// TIA Portal project "2022.11.26-双轴组合搬运" (V17)
// Vorlageprojekt für das Buch mit Zielsystem S7-1200

(* hardware
DEVICE "S7-1200-Station_1"  S7-1200 Station
   slot 0: "Baugruppenträger_0"  Rack  V1.0
   slot 1: "PLC_1"  CPU 1214C DC/DC/DC  6ES7 214-1AG40-0XB0  V4.5
*)

// ===== PLC "PLC_1"  CPU 1214C DC/DC/DC =====

VAR_GLOBAL   // PLC tag table "Standard-Variablentabelle"
   "启动" AT %I1.2 : Bool;
   "暂停" AT %I1.3 : Bool;
   "启动灯" AT %Q1.1 : Bool;
   "暂停2" AT %M10.1 : Bool;
   "暂停灯" AT %Q1.2 : Bool;
   "启动(1)" AT %M10.0 : Bool;
   "上升沿暂存位" AT %M100.0 : Bool;
   "生成器1" AT %Q1.3 : Bool;
   "生成器2" AT %Q1.4 : Bool;
   "传送带1" AT %Q0.3 : Bool;
   "传送带2" AT %Q0.6 : Bool;
   "感应器1" AT %I0.3 : Bool;
   "上升沿暂存位(1)" AT %M100.2 : Bool;
   "感应器2" AT %I0.6 : Bool;
   "缩回1" AT %Q0.4 : Bool;
   "缩回2" AT %Q0.7 : Bool;
   "上升沿暂存位（2）" AT %M100.3 : Bool;
   "Tag_1" AT %M100.1 : Bool;
   "下降沿暂存位（1）" AT %M100.4 : Bool;
   "下降沿暂存位（2）" AT %M100.5 : Bool;
   "缩回感应" AT %I0.4 : Bool;
   "缩回感应2" AT %I0.7 : Bool;
   "拿下降" AT %Q0.1 : Bool;
   "拿下降感应" AT %I0.1 : Bool;
   "拿吸" AT %Q0.2 : Bool;
   "拿吸感应" AT %I0.2 : Bool;
   "拿有物" AT %M10.2 : Bool;
   "拿伸出" AT %Q0.0 : Bool;
   "拿伸出感应" AT %I0.0 : Bool;
   "拿放中" AT %M10.3 : Bool;
   "完成放物" AT %M10.5 : Bool;
   "完成拿放" AT %M10.6 : Bool;
   "上升1" AT %Q0.5 : Bool;
   "上升2" AT %Q1.0 : Bool;
   "上升感应1" AT %I0.5 : Bool;
   "上升感应2" AT %I1.0 : Bool;
   "计数" AT %M10.7 : Bool;
   "下降沿暂存位" AT %M100.6 : Bool;
   "计数(1)" AT %QD30 : DWord;
   "数据清零" AT %I1.4 : Bool;
   "清零灯" AT %Q1.5 : Bool;
END_VAR

// folder: System blocks/Program resources

DATA_BLOCK "T0"   // DB1
{ S7_Optimized_Access := 'TRUE' }
AUTHOR : Simatic
FAMILY : IEC
NAME : IEC_TMR
VERSION : 1.0
// stored: InstanceOfName IEC_TIMER
"IEC_TIMER"
BEGIN
END_DATA_BLOCK

DATA_BLOCK "T1"   // DB2
{ S7_Optimized_Access := 'TRUE' }
AUTHOR : Simatic
FAMILY : IEC
NAME : IEC_TMR
VERSION : 1.0
// stored: InstanceOfName IEC_TIMER
"IEC_TIMER"
BEGIN
END_DATA_BLOCK

DATA_BLOCK "T2"   // DB3
{ S7_Optimized_Access := 'TRUE' }
AUTHOR : Simatic
FAMILY : IEC
NAME : IEC_TMR
VERSION : 1.0
// stored: InstanceOfName IEC_TIMER
"IEC_TIMER"
BEGIN
END_DATA_BLOCK

DATA_BLOCK "T3"   // DB4
{ S7_Optimized_Access := 'TRUE' }
AUTHOR : Simatic
FAMILY : IEC
NAME : IEC_TMR
VERSION : 1.0
// stored: InstanceOfName IEC_TIMER
"IEC_TIMER"
BEGIN
END_DATA_BLOCK

DATA_BLOCK "T4"   // DB5
{ S7_Optimized_Access := 'TRUE' }
AUTHOR : Simatic
FAMILY : IEC
NAME : IEC_TMR
VERSION : 1.0
// stored: InstanceOfName IEC_TIMER
"IEC_TIMER"
BEGIN
END_DATA_BLOCK

DATA_BLOCK "T5"   // DB6
{ S7_Optimized_Access := 'TRUE' }
AUTHOR : Simatic
FAMILY : IEC
NAME : IEC_TMR
VERSION : 1.0
// stored: InstanceOfName IEC_TIMER
"IEC_TIMER"
BEGIN
END_DATA_BLOCK

DATA_BLOCK "T6"   // DB7
{ S7_Optimized_Access := 'TRUE' }
AUTHOR : Simatic
FAMILY : IEC
NAME : IEC_TMR
VERSION : 1.0
// stored: InstanceOfName IEC_TIMER
"IEC_TIMER"
BEGIN
END_DATA_BLOCK

// folder: (top level)

FUNCTION "MHJ-PLC-Lab-Function-S71200" : Void   // FC9000, SCL
{ S7_Optimized_Access := 'TRUE' }
VERSION : 0.1
   VAR_TEMP
      rdTimeReturn : Int;
      outputTime : DTL;
      SyncVal : Byte;
      forVal : Int;
      forVal_2 : Int;
      Value : Byte;
   END_VAR
   VAR CONSTANT
      CompVal : Byte := 16#34;
      Value_01 : Byte := 16#11;
      Value_01_DW : DWord := 16#A165_D992;
      Value_02_DW : DWord := 16#58BE_4401;
   END_VAR
BEGIN

   #Value:=PEEK(area := 16#82,
        dbNumber := 0,
        byteOffset := 511);
   #Value := #Value + 1;

   POKE(area := 16#82,
        dbNumber := 0,
        byteOffset := 511,
        value := #Value);

   POKE(area:=16#81,
        dbNumber:=0,
        byteOffset:=1016,
        value:=#Value_01_DW);
   POKE(area := 16#81,
        dbNumber := 0,
        byteOffset := 1020,
        value := #Value_02_DW);

   POKE(area := 16#81,
        dbNumber := 0,
        byteOffset := 511,
        value := B#16#00);

   FOR #forVal := 0 TO 120 DO
       FOR #forVal_2:=0 TO 10 DO
           #rdTimeReturn:=RD_SYS_T(#outputTime);
           #rdTimeReturn := WR_SYS_T(#outputTime);
           #rdTimeReturn := RD_SYS_T(#outputTime);
           #rdTimeReturn := WR_SYS_T(#outputTime);
       END_FOR;
       #SyncVal:= PEEK(area := 16#81,
                      dbNumber := 0,
                      byteOffset := 511);
       IF #SyncVal = #CompVal THEN
          GOTO M_1;
       END_IF;
   END_FOR;
   RETURN;

   M_1:
   POKE(area := 16#81,
        dbNumber := 0,
        byteOffset := 511,
        value := B#16#0);
END_FUNCTION

ORGANIZATION_BLOCK "Main"   // OB1, LAD, ProgramCycle
TITLE = "Main Program Sweep (Cycle)"
{ S7_Optimized_Access := 'TRUE' }
VERSION : 0.1
   VAR_INPUT
      Initial_Call : Bool;   // Initial call of this OB
      Remanence : Bool;   // =True, if remanent data are available
   END_VAR
   VAR_TEMP   // added for the SCL form of the ladder/FBD networks
      _w1 : Bool;
      _w2 : Bool;
      _w3 : Bool;
      _w4 : Bool;
   END_VAR
BEGIN

REGION Network 1
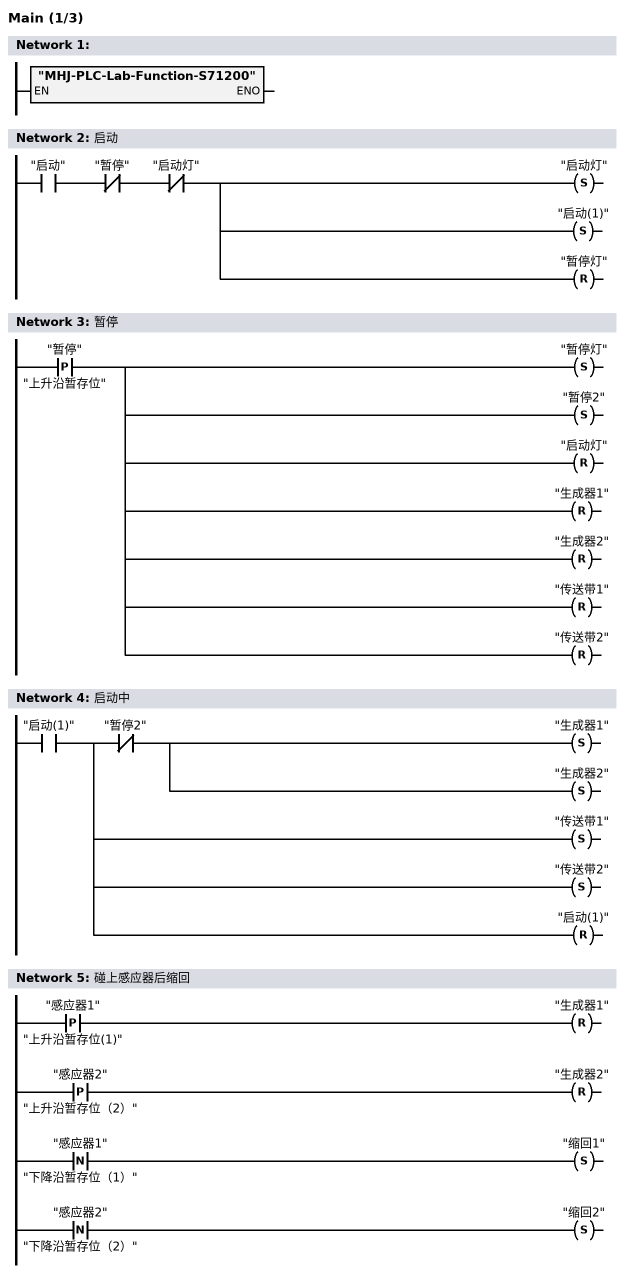
   RUNG wire#powerrail
      "MHJ-PLC-Lab-Function-S71200"()
   END_RUNG
   // the same network as SCL:
   "MHJ-PLC-Lab-Function-S71200"();
END_REGION

REGION Network 2: 启动
   RUNG wire#powerrail
      Contact( "启动" )
      I_Contact( "暂停" )
      I_Contact( "启动灯" )
      wire#w1
      S_Coil( "启动灯" )
   END_RUNG
   RUNG wire#w1
      S_Coil( "启动(1)" )
   END_RUNG
   RUNG wire#w1
      R_Coil( "暂停灯" )
   END_RUNG
   // the same network as SCL:
   #_w1 := "启动" AND NOT "暂停" AND NOT "启动灯";
   IF #_w1 THEN
       "启动灯" := TRUE;
       "启动(1)" := TRUE;
       "暂停灯" := FALSE;
   END_IF;
END_REGION

REGION Network 3: 暂停
   RUNG wire#powerrail
      P_Contact(operand := "暂停", bit := "上升沿暂存位")
      wire#w1
      S_Coil( "暂停灯" )
   END_RUNG
   RUNG wire#w1
      S_Coil( "暂停2" )
   END_RUNG
   RUNG wire#w1
      R_Coil( "启动灯" )
   END_RUNG
   RUNG wire#w1
      R_Coil( "生成器1" )
   END_RUNG
   RUNG wire#w1
      R_Coil( "生成器2" )
   END_RUNG
   RUNG wire#w1
      R_Coil( "传送带1" )
   END_RUNG
   RUNG wire#w1
      R_Coil( "传送带2" )
   END_RUNG
   // the same network as SCL:
   #_w1 := "暂停" AND NOT "上升沿暂存位";   // rising edge of "暂停"
   "上升沿暂存位" := "暂停";
   IF #_w1 THEN
       "暂停灯" := TRUE;
       "暂停2" := TRUE;
       "启动灯" := FALSE;
       "生成器1" := FALSE;
       "生成器2" := FALSE;
       "传送带1" := FALSE;
       "传送带2" := FALSE;
   END_IF;
END_REGION

REGION Network 4: 启动中
   RUNG wire#powerrail
      Contact( "启动(1)" )
      wire#w1
      I_Contact( "暂停2" )
      wire#w2
      S_Coil( "生成器1" )
   END_RUNG
   RUNG wire#w2
      S_Coil( "生成器2" )
   END_RUNG
   RUNG wire#w1
      S_Coil( "传送带1" )
   END_RUNG
   RUNG wire#w1
      S_Coil( "传送带2" )
   END_RUNG
   RUNG wire#w1
      R_Coil( "启动(1)" )
   END_RUNG
   // the same network as SCL:
   IF "启动(1)" AND NOT "暂停2" THEN
       "生成器1" := TRUE;
       "生成器2" := TRUE;
   END_IF;
   IF "启动(1)" THEN
       "传送带1" := TRUE;
       "传送带2" := TRUE;
       "启动(1)" := FALSE;
   END_IF;
END_REGION

REGION Network 5: 碰上感应器后缩回
   RUNG wire#powerrail
      P_Contact(operand := "感应器1", bit := "上升沿暂存位(1)")
      R_Coil( "生成器1" )
   END_RUNG
   RUNG wire#powerrail
      P_Contact(operand := "感应器2", bit := "上升沿暂存位（2）")
      R_Coil( "生成器2" )
   END_RUNG
   RUNG wire#powerrail
      N_Contact(operand := "感应器1", bit := "下降沿暂存位（1）")
      S_Coil( "缩回1" )
   END_RUNG
   RUNG wire#powerrail
      N_Contact(operand := "感应器2", bit := "下降沿暂存位（2）")
      S_Coil( "缩回2" )
   END_RUNG
   // the same network as SCL:
   #_w1 := "感应器1" AND NOT "上升沿暂存位(1)";   // rising edge of "感应器1"
   "上升沿暂存位(1)" := "感应器1";
   IF #_w1 THEN "生成器1" := FALSE; END_IF;
   #_w2 := "感应器2" AND NOT "上升沿暂存位（2）";   // rising edge of "感应器2"
   "上升沿暂存位（2）" := "感应器2";
   IF #_w2 THEN "生成器2" := FALSE; END_IF;
   #_w3 := NOT "感应器1" AND "下降沿暂存位（1）";   // falling edge of "感应器1"
   "下降沿暂存位（1）" := "感应器1";
   IF #_w3 THEN "缩回1" := TRUE; END_IF;
   #_w4 := NOT "感应器2" AND "下降沿暂存位（2）";   // falling edge of "感应器2"
   "下降沿暂存位（2）" := "感应器2";
   IF #_w4 THEN "缩回2" := TRUE; END_IF;
END_REGION

REGION Network 6: 缩回后拿下将
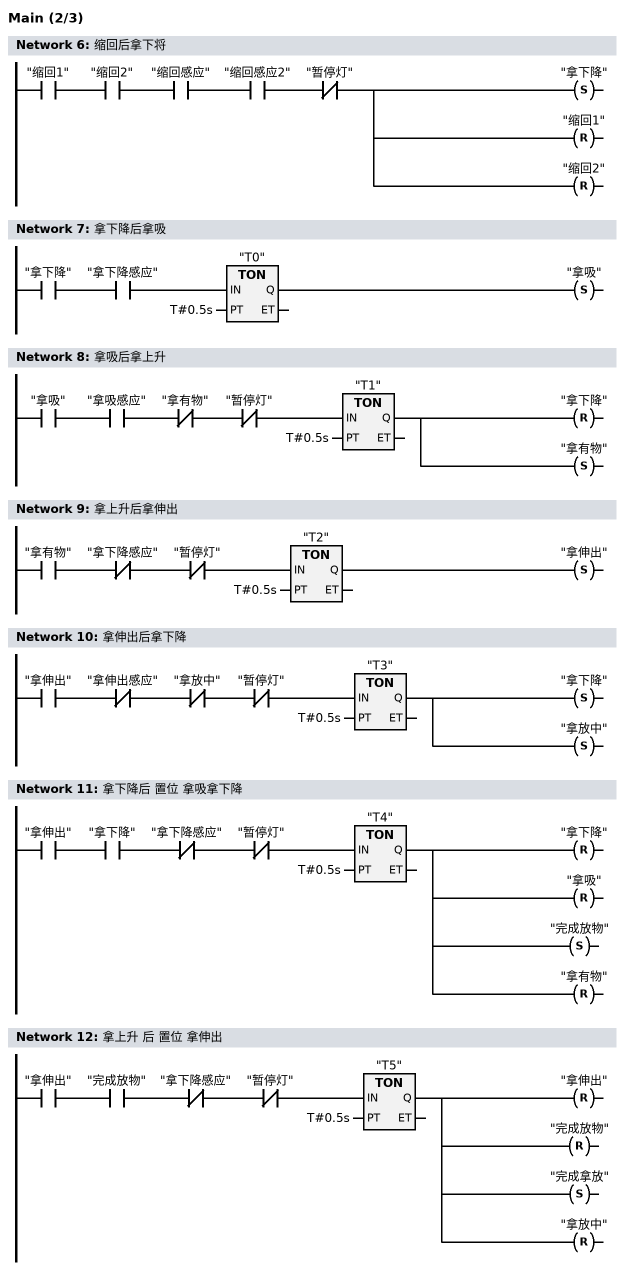
   RUNG wire#powerrail
      Contact( "缩回1" )
      Contact( "缩回2" )
      Contact( "缩回感应" )
      Contact( "缩回感应2" )
      I_Contact( "暂停灯" )
      wire#w1
      S_Coil( "拿下降" )
   END_RUNG
   RUNG wire#w1
      R_Coil( "缩回1" )
   END_RUNG
   RUNG wire#w1
      R_Coil( "缩回2" )
   END_RUNG
   // the same network as SCL:
   IF "缩回1" AND "缩回2" AND "缩回感应" AND "缩回感应2" AND NOT "暂停灯" THEN "拿下降" := TRUE; END_IF;
   #_w1 := "缩回1" AND "缩回2" AND "缩回感应" AND "缩回感应2" AND NOT "暂停灯";
   IF #_w1 THEN
       "缩回1" := FALSE;
       "缩回2" := FALSE;
   END_IF;
END_REGION

REGION Network 7: 拿下降后拿吸
   "T0".TON(IN := "拿下降" AND "拿下降感应", PT := T#0.5s);
   IF "T0".Q THEN "拿吸" := TRUE; END_IF;
END_REGION

REGION Network 8: 拿吸后拿上升
   "T1".TON(IN := "拿吸" AND "拿吸感应" AND NOT "拿有物" AND NOT "暂停灯", PT := T#0.5s);
   IF "T1".Q THEN
       "拿下降" := FALSE;
       "拿有物" := TRUE;
   END_IF;
END_REGION

REGION Network 9: 拿上升后拿伸出
   "T2".TON(IN := "拿有物" AND NOT "拿下降感应" AND NOT "暂停灯", PT := T#0.5s);
   IF "T2".Q THEN "拿伸出" := TRUE; END_IF;
END_REGION

REGION Network 10: 拿伸出后拿下降
   "T3".TON(IN := "拿伸出" AND NOT "拿伸出感应" AND NOT "拿放中" AND NOT "暂停灯", PT := T#0.5s);
   IF "T3".Q THEN
       "拿下降" := TRUE;
       "拿放中" := TRUE;
   END_IF;
END_REGION

REGION Network 11: 拿下降后 置位 拿吸拿下降
   "T4".TON(IN := "拿伸出" AND "拿下降" AND NOT "拿下降感应" AND NOT "暂停灯", PT := T#0.5s);
   IF "T4".Q THEN
       "拿下降" := FALSE;
       "拿吸" := FALSE;
       "完成放物" := TRUE;
       "拿有物" := FALSE;
   END_IF;
END_REGION

REGION Network 12: 拿上升 后 置位 拿伸出
   "T5".TON(IN := "拿伸出" AND "完成放物" AND NOT "拿下降感应" AND NOT "暂停灯", PT := T#0.5s);
   IF "T5".Q THEN
       "拿伸出" := FALSE;
       "完成放物" := FALSE;
       "完成拿放" := TRUE;
       "拿放中" := FALSE;
   END_IF;
END_REGION

REGION Network 13: 完成拿放挡上升
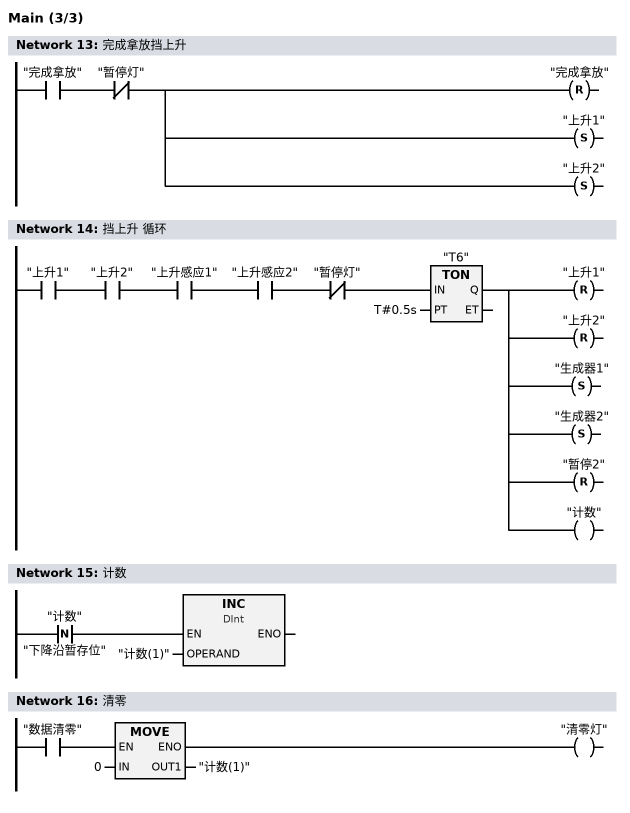
   RUNG wire#powerrail
      Contact( "完成拿放" )
      I_Contact( "暂停灯" )
      wire#w1
      R_Coil( "完成拿放" )
   END_RUNG
   RUNG wire#w1
      S_Coil( "上升1" )
   END_RUNG
   RUNG wire#w1
      S_Coil( "上升2" )
   END_RUNG
   // the same network as SCL:
   #_w1 := "完成拿放" AND NOT "暂停灯";
   IF #_w1 THEN
       "完成拿放" := FALSE;
       "上升1" := TRUE;
       "上升2" := TRUE;
   END_IF;
END_REGION

REGION Network 14: 挡上升 循环
   "T6".TON(IN := "上升1" AND "上升2" AND "上升感应1" AND "上升感应2" AND NOT "暂停灯", PT := T#0.5s);
   IF "T6".Q THEN
       "上升1" := FALSE;
       "上升2" := FALSE;
       "生成器1" := TRUE;
       "生成器2" := TRUE;
       "暂停2" := FALSE;
   END_IF;
   "计数" := "T6".Q;
END_REGION

REGION Network 15: 计数
   RUNG wire#powerrail
      N_Contact(operand := "计数", bit := "下降沿暂存位")
      { S7_Templates := "DestType := DInt" } Inc( "计数(1)" )
   END_RUNG
   // the same network as SCL:
   #_w1 := NOT "计数" AND "下降沿暂存位";   // falling edge of "计数"
   "下降沿暂存位" := "计数";
   IF #_w1 THEN "计数(1)" := "计数(1)" + 1; END_IF;
END_REGION

REGION Network 16: 清零
   RUNG wire#powerrail
      Contact( "数据清零" )
      Move(in := 0, out1 => "计数(1)")
      Coil( "清零灯" )
   END_RUNG
   // the same network as SCL:
   IF "数据清零" THEN "计数(1)" := 0; END_IF;
   "清零灯" := "数据清零";
END_REGION
END_ORGANIZATION_BLOCK